Yaskawa INFORM job: COPYVAR.JBI

/JOB
//NAME COPYVAR
///FOLDERNAME IMPORTANT_JOBS
//POS
///NPOS 0,0,0,2,0,0
///TOOL 0
///POSTYPE BASE
///RECTAN
///RCONF 1,0,0,0,0,0,0,0,0,0,0,0,0,0,0,0,0,0,0,0,0,0,0,0
P00301=0.046,-2.112,7.779,0.0000,0.0000,0.0000
P00302=-0.180,-2.409,6.326,0.0000,0.0000,0.0000
//INST
///DATE 2024/04/16 08:57
///ATTR SC,RW
///GROUP1 RB1,BS1
NOP
GETE D040 P0301 (1)
GETE D041 P0301 (2)
GETE D042 P0301 (3)
SETE P0302 (1) D040
SETE P0302 (2) D041
SETE P0302 (3) D042
END
